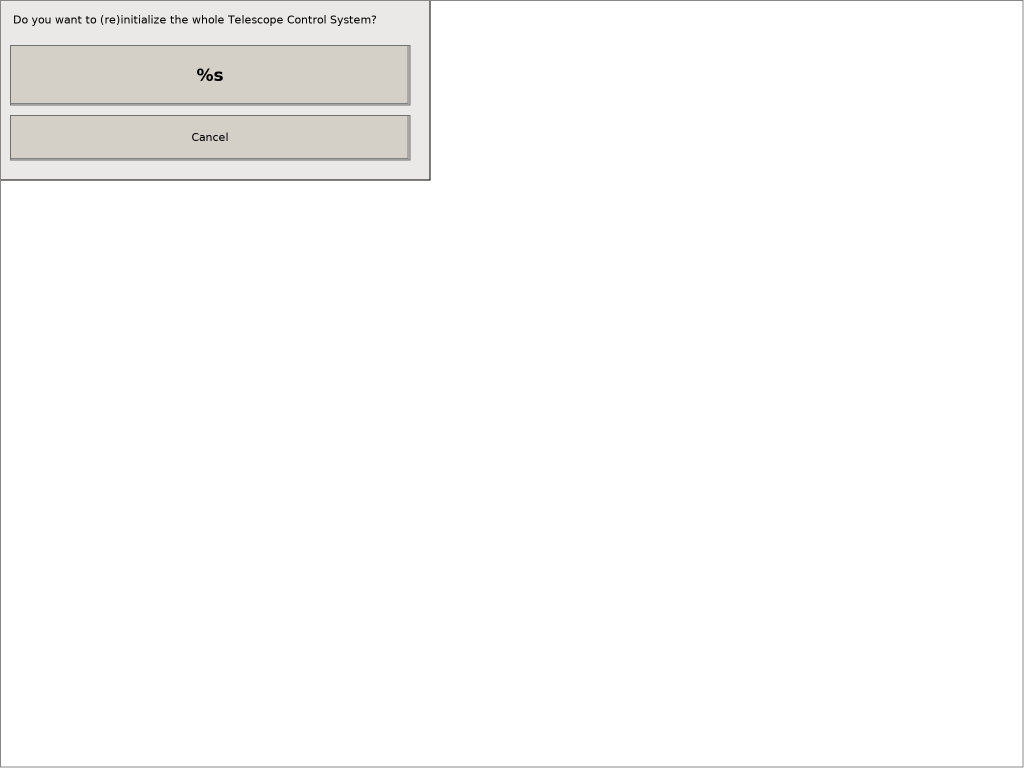
VISUALIZATION VISU_MTCSInitializeDialog  // 1024x768
    Rectangle (0,0 430x180)
    Button (10,115 400x45), "Cancel"
        OnMouseClick: CloseDialog Dialog=VISU_MTCSInitializeDialog, Result=OK, NumpadKeypadSet=True
    Label (10,5 400x30), "Do you want to (re)initialize the whole Telescope Control System?"
    Button (10,45 400x60), "%s", text variable: GLOBAL.gui.button_initialize.textOneLine, input disabled if: GLOBAL.gui.button_initialize.deactivate
        OnMouseClick: execute { GLOBAL.gui.button_initialize.do_request := TRUE; }
        OnMouseClick: CloseDialog Dialog=VISU_MTCSInitializeDialog, Result=OK, NumpadKeypadSet=True
END_VISUALIZATION

(* stored: Version 1.1.0.1, ProductVersion 3.1.4018.5
   Visu VISU_MTCSInitializeDialog: Id {c6cb8c68-f106-44e6-8826-952f68c1d482} *)
